PROGRAM MAIN
VAR		
	bStartProcess 	: BOOL := FALSE;
	timer1			: TON;
	timer2			: TON;
	timer3			: TON;
	bStart1			: BOOL := FALSE;
	bStart2: BOOL;
	bStart3: BOOL;
END_VAR

// Beginning of painting process //

// If process is initiated from UI
IF (bStartProcess) THEN
	bStart1 := TRUE;
	timer1(IN := bStart1, PT:= T#5S);
		
	IF timer1.Q THEN		
		Variables.nFANUC_REMOTE_START := 160; // Initializing variables #6 (Starts)
		bStart2 := TRUE;
	END_IF
	
	COMM_FANUC.arrf_Internal_FANUC_Output_1 := 63; // Tell FANUC to move and leave robot in initial position	
	
	timer2(IN := bStart2, PT:= T#1S);
		
	IF timer2.Q THEN		
		Variables.nFANUC_REMOTE_START := 128; // Start works in a rising edge
	END_IF
	
	
	IF COMM_FANUC.arrf_Internal_FANUC_Input_1 = 254 THEN // IF FANUC tells us that position has been reached, we proceed to move UR
		Variables.nURProgAction := 63; // Set Program in UR - Move Robot		
		// Wait for UR to finish
		
		IF Variables.nURProgState = 99 THEN // If UR finishes
			COMM_FANUC.arrf_Internal_FANUC_Output_1 := 77; // Inform FANUC that it is safe to move home
			bStart3 := TRUE;			
			timer3(IN := bStart3, PT:= T#3S);			
			IF timer3.Q THEN
				
				bStartProcess := FALSE; // Terminate process
			END_IF
								
		END_IF		
	END_IF

ELSE // IF not initiated
	// While no signal for starting demo is coming, set variables of robots as 0
	//timer1.IN := FALSE;
	//Variables.nFANUC_REMOTE_START := 0;
	COMM_FANUC.arrf_Internal_FANUC_Output_1 := 0;
	Variables.nURProgAction := 0;
	Variables.nFANUC_REMOTE_START := 128; // Initializing variables #8 (Enable function)
	bStart1 := FALSE;
	bStart2 := FALSE;
	bStart3 := FALSE;
	timer1(IN:=bStart1);
	timer2(IN:=bStart2);
	timer3(IN:=bStart3);
END_IF


Data_Publisher();
COMM_UR10();
COMM_FANUC();
Analog_Speed();

END_PROGRAM

(* stored: Version 1.1.0.1, ProductVersion 3.1.4024.0
   POU MAIN: Id {acd9ff64-481e-460e-9be1-ced6f2e40b6e}, SpecialFunc None *)
